// SIMATIC S7-200 project (STEP 7-Micro/WIN), CPU 221 REL 01.10

ORGANIZATION_BLOCK 主程序:OB1
TITLE=程序注释
BEGIN
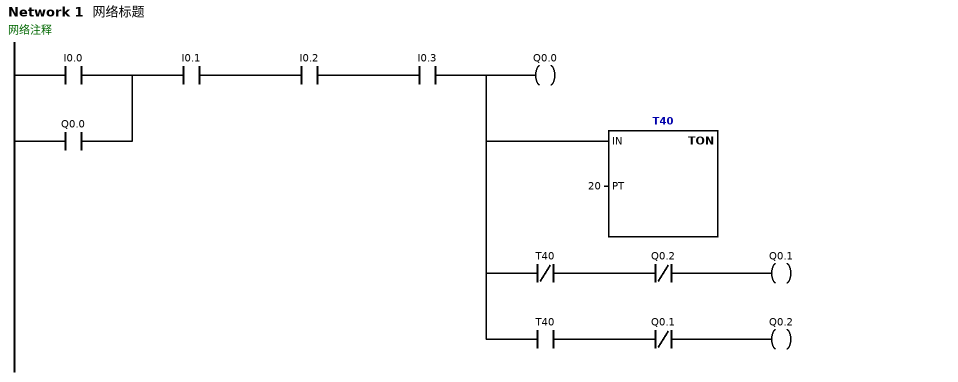
Network 1 // 网络标题
// 网络注释
LD     I0.0
O      Q0.0
A      I0.1
A      I0.2
A      I0.3
LPS
=      Q0.0
TON    T40, 20
AN     T40
AN     Q0.2
=      Q0.1
LPP
A      T40
AN     Q0.1
=      Q0.2
END_ORGANIZATION_BLOCK
